Universal Robots PolyScope program: Test ur5.urp

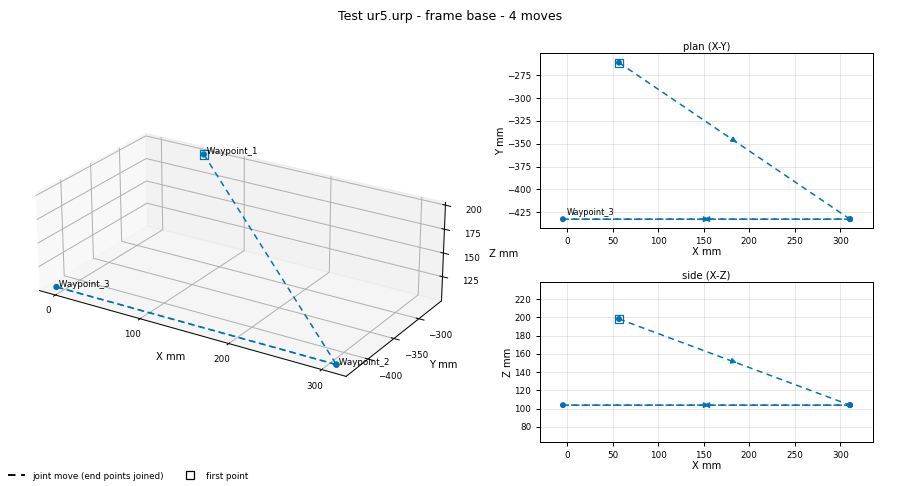
[picture p0: tool path of Test ur5.urp in frame base, 4 of 4 moves have a stored position in this frame; points joined in program order, loops and branches not executed]
Program Test ur5 (installation=default directory=/programs/usbdisk/NoodleBotSoftware createdIn=3.12.1.90940 lastSavedIn=3.12.1.90940 robotSerialNumber=2017354841)
Calibrated DH parameters: a=[0.000094, -0.006117, -0.382762, 0.000086, 0.000044, 0]; d=[0.089236, 217.751846, -204.357806, -13.283746, 0.094902, 0.082641]; alpha=[1.57017, 0.001953, -0.006493, 1.570192, -1.570543, 0]; deltaTheta=[0.000036, 1.556386, -1.779789, 0.223359, -0.000014, -0.000001]
Robot Program (runOnlyOnce=false)
  MoveJ speed 60 deg/s, acceleration 80 deg/s^2 (useActiveTCP=true)
    Waypoint Waypoint_1: TCP in base x=56.966 y=-261.001 z=198.306 mm, rx=1.7335 ry=1.785 rz=-0.8303 rad; joints [88.749, -149.236, 145.835, 226.397, 267.6, 85.926] deg; flange x=103.365 y=-153.635 z=343.802 mm, rx=1.7335 ry=1.785 rz=-0.8304 rad
    Wait Sleep waitTime=1
    Waypoint Waypoint_2: TCP in base x=310.686 y=-432.811 z=103.702 mm, rx=2.1474 ry=-0.8604 rz=-0.3969 rad; joints [132.489, -81.812, 115.29, 232.118, 220.576, -95.949] deg; flange x=364.062 y=-326.662 z=247.669 mm, rx=2.1474 ry=-0.8605 rz=-0.3969 rad
    Wait Sleep waitTime=1
    Waypoint Waypoint_3: TCP in base x=-4.542 y=-432.806 z=103.696 mm, rx=2.1474 ry=-0.8605 rz=-0.397 rad; joints [86.389, -101.139, 144.341, 185.043, 240.669, -151.599] deg; flange x=48.86 y=-326.662 z=247.669 mm, rx=2.1474 ry=-0.8605 rz=-0.3969 rad
    Wait Sleep waitTime=1
    Waypoint Waypoint_2: TCP in base x=310.686 y=-432.811 z=103.702 mm, rx=2.1474 ry=-0.8604 rz=-0.3969 rad; joints [132.489, -81.812, 115.29, 232.118, 220.576, -95.949] deg; flange x=364.062 y=-326.662 z=247.669 mm, rx=2.1474 ry=-0.8605 rz=-0.3969 rad
